{attribute 'qualified_only'}
{attribute 'strict'}
TYPE E_RobotClamp :
(
	ClampA := 1,
	ClampB
);
END_TYPE

(* stored: Version 1.1.0.1, ProductVersion 3.1.4024.13
   DUT E_RobotClamp: Id {e125f21e-2366-4c9a-a2f0-81d067862af6} *)
